FUNCTION_BLOCK FB_Hysteresis
VAR_INPUT
	In: REAL;
	On_val: REAL;
	Off_val: REAL;
END_VAR
VAR_OUTPUT
	Out: BOOL;
END_VAR
VAR	
END_VAR

IF In > On_val THEN
	Out:= TRUE;
END_IF
IF In < Off_val THEN
	Out:= FALSE;
END_IF

END_FUNCTION_BLOCK

(* stored: Version 1.1.0.1, ProductVersion 3.1.4024.0
   POU FB_Hysteresis: Id {9ab13096-d9d9-4d3a-80dd-5708fa4e5ce0}, SpecialFunc None *)
